(* PLC project PLC, Beckhoff Automation GmbH TwinCAT PLC Control 3.5.13.21 *)
(* stored: creationDateTime 2024-02-17T22:43:01.2031282, modificationDateTime 2024-02-17T22:43:01.2031282 *)

TYPE CylStatus :
STRUCT
	name: STRING(G.nameStringLength);
	opeFw: BOOL;
	opeRv: BOOL;
	posFw: BOOL;
	posRv: BOOL;
	ready: BOOL;
	busy: BOOL;
	done: BOOL;
	error: BOOL;
	errorCode: LINT;
	opePastTime: TIME;
END_STRUCT
END_TYPE
